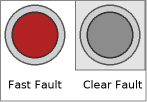
VISUALIZATION FastFaultGUI  // 147x102
VAR_IN_OUT
	FastFault	:	FB_HardwareFFOutput;
END_VAR
    Lamp1 (0,0 70x70), variable: NOT FastFault.q_xFastFaultOut, style: Lamp-Lamp1-Red
    Label (5,70 59x30), "Fast Fault"
    PushSwitch (75,0 70x70), variable: FastFault.i_xReset, behaviour: TAP, style: Switch-PushSwitch-Gray
    Label (80,70 59x30), "Clear Fault"
END_VISUALIZATION

(* stored: Version 1.1.0.1, ProductVersion 3.1.4022.12
   Visu FastFaultGUI: Id {db6c9ea9-b8b7-0c47-0a09-029526e91248} *)
